INTERFACE I_OutputPortVisitor

METHOD VisitOutputPort
VAR_INPUT
	VisitingOutputPort : I_OutputPort;
END_VAR
END_METHOD

END_INTERFACE

(* stored: Version 1.1.0.1, ProductVersion 3.1.4024.12
   Itf I_OutputPortVisitor: Id {0a4111b2-dfa4-09fe-37bf-80540c755e7a}
   Method VisitOutputPort: Id {a7212b88-253f-0d9b-3231-b721ab280805} *)
